TYPE MC_COMMAND_REF :
STRUCT
	CommandId : INT;
END_STRUCT
END_TYPE

(* stored: Version 1.1.0.1, ProductVersion 3.1.4024.11
   DUT MC_COMMAND_REF: Id {c7ffce84-6a3a-4708-8a13-ff285a83f9c0} *)
